PROGRAM MAIN
VAR CONSTANT
END_VAR
VAR
	ulimit	:	DINT	:=	1000;
	delay	:	DINT	:=	50;
	assign	:	BOOL	:=	FALSE;
	(**********************)
	arr	:	ARRAY	[0..20000]	OF	iterator;
	cache	:	ARRAY	[0..20000]	OF	DINT;
	noToTest	:	DINT	:= 0;
	count	: DINT	:=0;
	I	:	DINT;
	step	:	BOOL;
END_VAR


IF count < delay-1 THEN
	count := count + 1;
	step :=	FALSE;
ELSE
	count := 0;
	step :=	TRUE;
END_IF

IF step THEN
	IF noToTest < ulimit-1 THEN
		noToTest := noToTest + 1;
	ELSE
		noToTest := 0;
	END_IF
END_IF
// Run noToTest operations
FOR I:=0 TO noToTest BY 1 DO 
	arr[I](increment:=1);
	IF ASSIGN THEN
		cache[I] := arr[i].out;
	END_IF
END_FOR;

END_PROGRAM

(* stored: Version 1.1.0.1, ProductVersion 3.1.4020.12
   POU MAIN: Id {e0313068-1eb6-4e3d-8bcd-3e27c74f9e5d}, SpecialFunc None *)
